// TIA Portal project "Projec1214" (V17)

(* hardware
DEVICE "S7-1200 station_1"  S7-1200 Station
   slot 0: "Rack_0"  S7-1200 Rack  Rack  V1.0
   slot 1: "PLC_1"  CPU 1211C DC/DC/Rly  6ES7 211-1HE40-0XB0  V4.5
DEVICE "HMI_1"  KTP400 Comfort
   slot 0: "HMI_1"  KTP400 Comfort  6AV2 124-2DC01-0AX0  17.0.0.0
   slot 1: "HMI_RT_1"  KTP400 Comfort  6AV2 124-2DC01-0AX0  17.0.0.0
   slot 5: "HMI_1.IE_CP_1"  PROFINET Interface  17.0.0.0
      slot 1: "PROFINET Interface_1"  PROFINET Interface
         slot 1: "Port_1"  Port
   slot 7: "HMI_1.MPI/DP_CP_1"  MPI/DP Interface  17.0.0.0
*)

// ===== PLC "PLC_1"  CPU 1211C DC/DC/Rly =====

VAR_GLOBAL   // PLC tag table "Default tag table"
   "BP_Appel_ET1" AT %I0.1 : Bool;
   "BP_Appel_ET2" AT %I0.2 : Bool;
   "BP_Appel_ET3" AT %I0.3 : Bool;
   "Position_ET1" AT %I0.5 : Bool;
   "Position_ET2" AT %I0.6 : Bool;
   "Position_ET3" AT %I0.7 : Bool;
   "Monter" AT %Q0.0 : Bool;
   "Descente" AT %Q0.1 : Bool;
   "Ouverture" AT %Q0.2 : Bool;
   "Fermeture" AT %Q0.3 : Bool;
   "MemoAppelET1" AT %M10.1 : Bool;
   "MemoAppelET2" AT %M10.2 : Bool;
   "MemoAppelET3" AT %M10.3 : Bool;
   "ETAPE0" AT %M10.4 : Bool;
   "ETAPE1" AT %M10.5 : Bool;
   "ETAPE2" AT %M10.6 : Bool;
   "ETAPE3" AT %M10.7 : Bool;
   "ETAPE4" AT %M11.0 : Bool;
   "ETAPE5" AT %M11.1 : Bool;
   "ETAPE6" AT %M11.2 : Bool;
   "ETAPE7" AT %M11.3 : Bool;
   "ETAPE8" AT %M11.4 : Bool;
   "ETAPE9" AT %M11.5 : Bool;
   "PorteOuverte" AT %I1.0 : Bool;
   "PorteFermee" AT %I1.1 : Bool;
   "MemoPosiET1" AT %M11.6 : Bool;
   "MemoPosiET2" AT %M11.7 : Bool;
   "MemoPosiET3" AT %M12.0 : Bool;
   "MemoPorteOuverte" AT %M12.1 : Bool;
   "MemoPorteFermee" AT %M12.2 : Bool;
   "DemandeNiveau1" AT %M40.0 : Bool;
   "DemandeNIveau2" AT %M40.1 : Bool;
   "DemandeNiveau3" AT %M40.2 : Bool;
   "Tag_4" AT %M40.3 : Bool;
   "Tag_5" AT %M40.4 : Bool;
   "Tag_6" AT %M40.5 : Bool;
   "Tag_7" AT %M40.6 : Bool;
   "Tag_8" AT %M40.7 : Bool;
   "deplacemntAsceseur" AT %MW100 : Int;
   "DeplacementPorteG" AT %MW102 : Int;
   "DeplacementPorteD" AT %MW104 : Int;
   "Clock_Byte" AT %MB0 : Byte;
   "Clock_10Hz" AT %M0.0 : Bool;
   "Clock_5Hz" AT %M0.1 : Bool;
   "Clock_2.5Hz" AT %M0.2 : Bool;
   "Clock_2Hz" AT %M0.3 : Bool;
   "Clock_1.25Hz" AT %M0.4 : Bool;
   "Clock_1Hz" AT %M0.5 : Bool;
   "Clock_0.625Hz" AT %M0.6 : Bool;
   "Clock_0.5Hz" AT %M0.7 : Bool;
   "deplacementHautPorte" AT %MW106 : Int;
END_VAR

DATA_BLOCK "ETAPE"   // DB1
{ S7_Optimized_Access := 'TRUE' }
VERSION : 0.1
   VAR
      "1" : Bool;
      "0" : Bool;
      "2" : Bool;
      "3" : Bool;
      "6" : Bool;
      "7" : Bool;
      "8" : Bool;
   END_VAR
BEGIN
END_DATA_BLOCK

// folder: System blocks/Program resources

DATA_BLOCK "IEC_Timer_0_DB"   // DB2
{ S7_Optimized_Access := 'TRUE' }
AUTHOR : Simatic
FAMILY : IEC
NAME : IEC_TMR
VERSION : 1.0
// stored: InstanceOfName IEC_TIMER
"IEC_TIMER"
BEGIN
END_DATA_BLOCK

// folder: (top level)

ORGANIZATION_BLOCK "Main"   // OB1, LAD, ProgramCycle
TITLE = "Main Program Sweep (Cycle)"
{ S7_Optimized_Access := 'TRUE' }
VERSION : 0.1
   VAR_INPUT
      Initial_Call : Bool;   // Initial call of this OB
      Remanence : Bool;   // =True, if remanent data are available
   END_VAR
   VAR_TEMP   // added for the SCL form of the ladder/FBD networks
      _w1 : Bool;
   END_VAR
BEGIN

REGION Network 1: ETAPE0
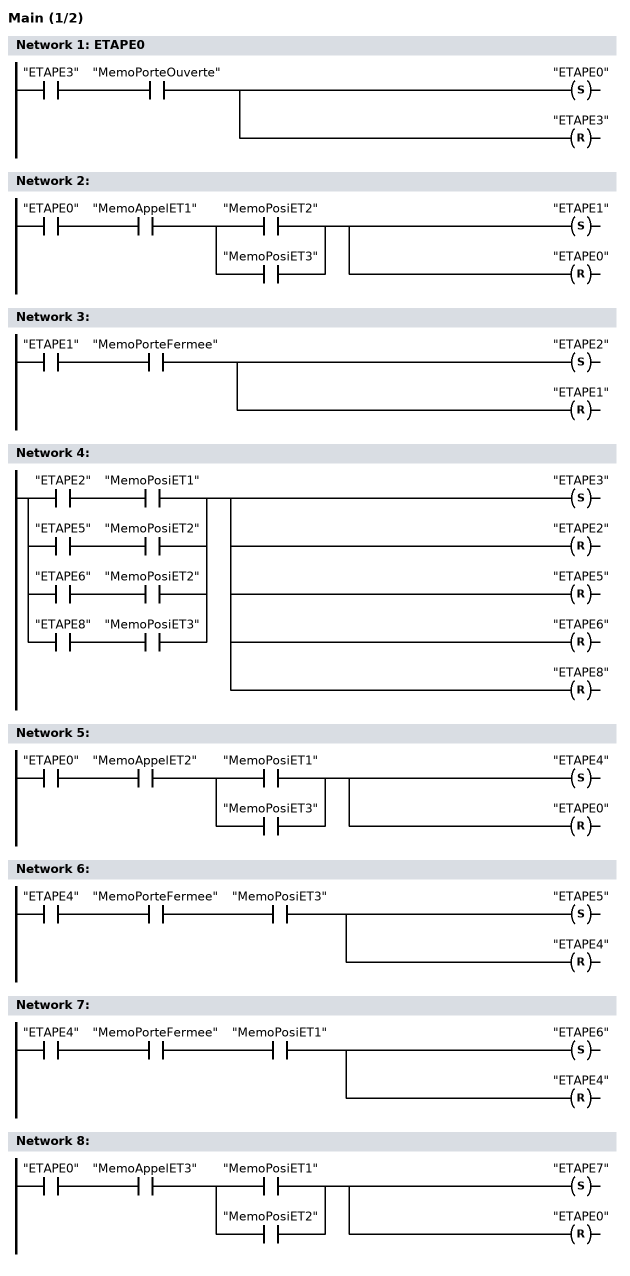
   RUNG wire#powerrail
      Contact( "ETAPE3" )
      Contact( "MemoPorteOuverte" )
      wire#w1
      S_Coil( "ETAPE0" )
   END_RUNG
   RUNG wire#w1
      R_Coil( "ETAPE3" )
   END_RUNG
   // the same network as SCL:
   IF "ETAPE3" AND "MemoPorteOuverte" THEN
       "ETAPE0" := TRUE;
       "ETAPE3" := FALSE;
   END_IF;
END_REGION

REGION Network 2
   RUNG wire#powerrail
      Contact( "ETAPE0" )
      Contact( "MemoAppelET1" )
      wire#w1
      Contact( "MemoPosiET2" )
      wire#w2
      S_Coil( "ETAPE1" )
   END_RUNG
   RUNG wire#w1
      Contact( "MemoPosiET3" )
   END_RUNG wire#w2
   RUNG wire#w2
      R_Coil( "ETAPE0" )
   END_RUNG
   // the same network as SCL:
   IF "ETAPE0" AND "MemoAppelET1" AND ("MemoPosiET2" OR "MemoPosiET3") THEN
       "ETAPE1" := TRUE;
       "ETAPE0" := FALSE;
   END_IF;
END_REGION

REGION Network 3
   RUNG wire#powerrail
      Contact( "ETAPE1" )
      Contact( "MemoPorteFermee" )
      wire#w1
      S_Coil( "ETAPE2" )
   END_RUNG
   RUNG wire#w1
      R_Coil( "ETAPE1" )
   END_RUNG
   // the same network as SCL:
   IF "ETAPE1" AND "MemoPorteFermee" THEN
       "ETAPE2" := TRUE;
       "ETAPE1" := FALSE;
   END_IF;
END_REGION

REGION Network 4
   RUNG wire#powerrail
      Contact( "ETAPE2" )
      Contact( "MemoPosiET1" )
      wire#w1
      S_Coil( "ETAPE3" )
   END_RUNG
   RUNG wire#powerrail
      Contact( "ETAPE5" )
      Contact( "MemoPosiET2" )
   END_RUNG wire#w1
   RUNG wire#powerrail
      Contact( "ETAPE6" )
      Contact( "MemoPosiET2" )
   END_RUNG wire#w1
   RUNG wire#powerrail
      Contact( "ETAPE8" )
      Contact( "MemoPosiET3" )
   END_RUNG wire#w1
   RUNG wire#w1
      R_Coil( "ETAPE2" )
   END_RUNG
   RUNG wire#w1
      R_Coil( "ETAPE5" )
   END_RUNG
   RUNG wire#w1
      R_Coil( "ETAPE6" )
   END_RUNG
   RUNG wire#w1
      R_Coil( "ETAPE8" )
   END_RUNG
   // the same network as SCL:
   IF ("ETAPE2" AND "MemoPosiET1") OR ("ETAPE5" AND "MemoPosiET2") OR ("ETAPE6" AND "MemoPosiET2") OR ("ETAPE8" AND "MemoPosiET3") THEN
       "ETAPE3" := TRUE;
   END_IF;
   #_w1 := ("ETAPE2" AND "MemoPosiET1") OR ("ETAPE5" AND "MemoPosiET2") OR ("ETAPE6" AND "MemoPosiET2") OR ("ETAPE8" AND "MemoPosiET3");
   IF #_w1 THEN
       "ETAPE2" := FALSE;
       "ETAPE5" := FALSE;
       "ETAPE6" := FALSE;
       "ETAPE8" := FALSE;
   END_IF;
END_REGION

REGION Network 5
   RUNG wire#powerrail
      Contact( "ETAPE0" )
      Contact( "MemoAppelET2" )
      wire#w1
      Contact( "MemoPosiET1" )
      wire#w2
      S_Coil( "ETAPE4" )
   END_RUNG
   RUNG wire#w1
      Contact( "MemoPosiET3" )
   END_RUNG wire#w2
   RUNG wire#w2
      R_Coil( "ETAPE0" )
   END_RUNG
   // the same network as SCL:
   IF "ETAPE0" AND "MemoAppelET2" AND ("MemoPosiET1" OR "MemoPosiET3") THEN
       "ETAPE4" := TRUE;
       "ETAPE0" := FALSE;
   END_IF;
END_REGION

REGION Network 6
   RUNG wire#powerrail
      Contact( "ETAPE4" )
      Contact( "MemoPorteFermee" )
      Contact( "MemoPosiET3" )
      wire#w1
      S_Coil( "ETAPE5" )
   END_RUNG
   RUNG wire#w1
      R_Coil( "ETAPE4" )
   END_RUNG
   // the same network as SCL:
   IF "ETAPE4" AND "MemoPorteFermee" AND "MemoPosiET3" THEN
       "ETAPE5" := TRUE;
       "ETAPE4" := FALSE;
   END_IF;
END_REGION

REGION Network 7
   RUNG wire#powerrail
      Contact( "ETAPE4" )
      Contact( "MemoPorteFermee" )
      Contact( "MemoPosiET1" )
      wire#w1
      S_Coil( "ETAPE6" )
   END_RUNG
   RUNG wire#w1
      R_Coil( "ETAPE4" )
   END_RUNG
   // the same network as SCL:
   IF "ETAPE4" AND "MemoPorteFermee" AND "MemoPosiET1" THEN
       "ETAPE6" := TRUE;
       "ETAPE4" := FALSE;
   END_IF;
END_REGION

REGION Network 8
   RUNG wire#powerrail
      Contact( "ETAPE0" )
      Contact( "MemoAppelET3" )
      wire#w1
      Contact( "MemoPosiET1" )
      wire#w2
      S_Coil( "ETAPE7" )
   END_RUNG
   RUNG wire#w1
      Contact( "MemoPosiET2" )
   END_RUNG wire#w2
   RUNG wire#w2
      R_Coil( "ETAPE0" )
   END_RUNG
   // the same network as SCL:
   IF "ETAPE0" AND "MemoAppelET3" AND ("MemoPosiET1" OR "MemoPosiET2") THEN
       "ETAPE7" := TRUE;
       "ETAPE0" := FALSE;
   END_IF;
END_REGION

REGION Network 9
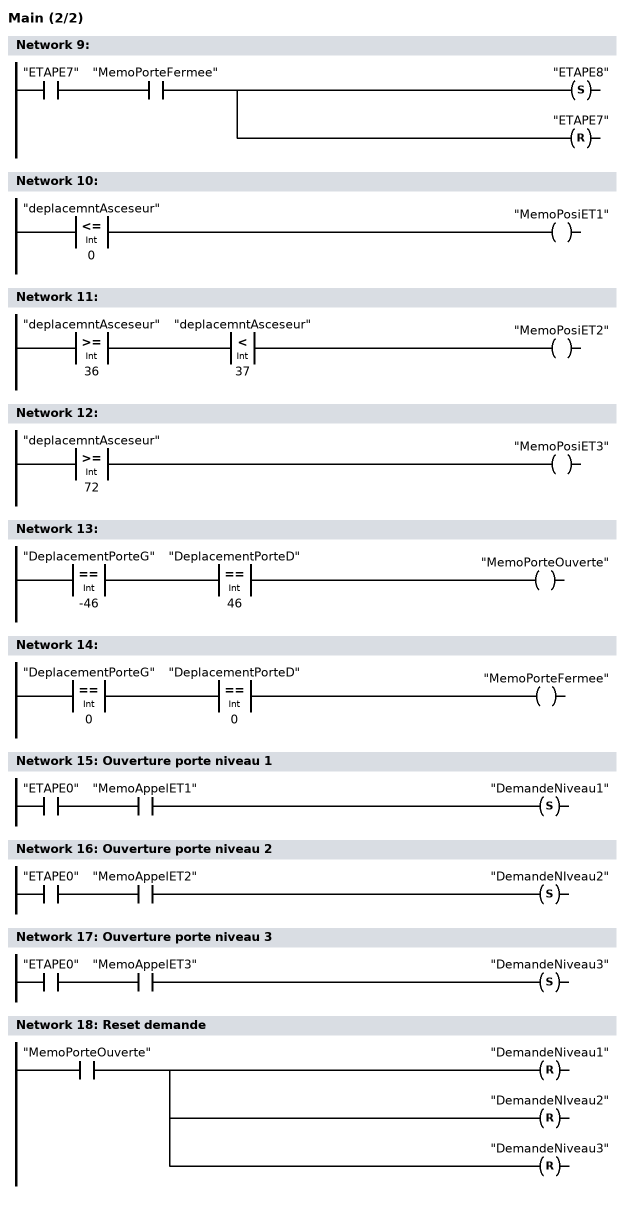
   RUNG wire#powerrail
      Contact( "ETAPE7" )
      Contact( "MemoPorteFermee" )
      wire#w1
      S_Coil( "ETAPE8" )
   END_RUNG
   RUNG wire#w1
      R_Coil( "ETAPE7" )
   END_RUNG
   // the same network as SCL:
   IF "ETAPE7" AND "MemoPorteFermee" THEN
       "ETAPE8" := TRUE;
       "ETAPE7" := FALSE;
   END_IF;
END_REGION

REGION Network 10
   RUNG wire#powerrail
      { S7_Templates := "SrcType := Int" } LE_Contact(in1 := "deplacemntAsceseur", in2 := 0)
      Coil( "MemoPosiET1" )
   END_RUNG
   // the same network as SCL:
   "MemoPosiET1" := "deplacemntAsceseur" <= 0;
END_REGION

REGION Network 11
   RUNG wire#powerrail
      { S7_Templates := "SrcType := Int" } GE_Contact(in1 := "deplacemntAsceseur", in2 := 36)
      { S7_Templates := "SrcType := Int" } LT_Contact(in1 := "deplacemntAsceseur", in2 := 37)
      Coil( "MemoPosiET2" )
   END_RUNG
   // the same network as SCL:
   "MemoPosiET2" := ("deplacemntAsceseur" >= 36) AND ("deplacemntAsceseur" < 37);
END_REGION

REGION Network 12
   RUNG wire#powerrail
      { S7_Templates := "SrcType := Int" } GE_Contact(in1 := "deplacemntAsceseur", in2 := 72)
      Coil( "MemoPosiET3" )
   END_RUNG
   // the same network as SCL:
   "MemoPosiET3" := "deplacemntAsceseur" >= 72;
END_REGION

REGION Network 13
   RUNG wire#powerrail
      { S7_Templates := "SrcType := Int" } EQ_Contact(in1 := "DeplacementPorteG", in2 := -46)
      { S7_Templates := "SrcType := Int" } EQ_Contact(in1 := "DeplacementPorteD", in2 := 46)
      Coil( "MemoPorteOuverte" )
   END_RUNG
   // the same network as SCL:
   "MemoPorteOuverte" := ("DeplacementPorteG" = (-46)) AND ("DeplacementPorteD" = 46);
END_REGION

REGION Network 14
   RUNG wire#powerrail
      { S7_Templates := "SrcType := Int" } EQ_Contact(in1 := "DeplacementPorteG", in2 := 0)
      { S7_Templates := "SrcType := Int" } EQ_Contact(in1 := "DeplacementPorteD", in2 := 0)
      Coil( "MemoPorteFermee" )
   END_RUNG
   // the same network as SCL:
   "MemoPorteFermee" := ("DeplacementPorteG" = 0) AND ("DeplacementPorteD" = 0);
END_REGION

REGION Network 15: Ouverture porte niveau 1
   RUNG wire#powerrail
      Contact( "ETAPE0" )
      Contact( "MemoAppelET1" )
      S_Coil( "DemandeNiveau1" )
   END_RUNG
   // the same network as SCL:
   IF "ETAPE0" AND "MemoAppelET1" THEN "DemandeNiveau1" := TRUE; END_IF;
END_REGION

REGION Network 16: Ouverture porte niveau 2
   RUNG wire#powerrail
      Contact( "ETAPE0" )
      Contact( "MemoAppelET2" )
      S_Coil( "DemandeNIveau2" )
   END_RUNG
   // the same network as SCL:
   IF "ETAPE0" AND "MemoAppelET2" THEN "DemandeNIveau2" := TRUE; END_IF;
END_REGION

REGION Network 17: Ouverture porte niveau 3
   RUNG wire#powerrail
      Contact( "ETAPE0" )
      Contact( "MemoAppelET3" )
      S_Coil( "DemandeNiveau3" )
   END_RUNG
   // the same network as SCL:
   IF "ETAPE0" AND "MemoAppelET3" THEN "DemandeNiveau3" := TRUE; END_IF;
END_REGION

REGION Network 18: Reset demande
   RUNG wire#powerrail
      Contact( "MemoPorteOuverte" )
      wire#w1
      R_Coil( "DemandeNiveau1" )
   END_RUNG
   RUNG wire#w1
      R_Coil( "DemandeNIveau2" )
   END_RUNG
   RUNG wire#w1
      R_Coil( "DemandeNiveau3" )
   END_RUNG
   // the same network as SCL:
   IF "MemoPorteOuverte" THEN
       "DemandeNiveau1" := FALSE;
       "DemandeNIveau2" := FALSE;
       "DemandeNiveau3" := FALSE;
   END_IF;
END_REGION
END_ORGANIZATION_BLOCK

ORGANIZATION_BLOCK "Cyclic interrupt"   // OB30, LAD, CyclicInterrupt
{ S7_Optimized_Access := 'TRUE' }
VERSION : 0.1
   VAR_INPUT
      Initial_Call : Bool;   // Initial call of this OB
      Event_Count : Int;   // Events discarded
   END_VAR
   VAR_TEMP   // added for the SCL form of the ladder/FBD networks
      _w1 : Bool;
   END_VAR
BEGIN

REGION Network 1: Fermeture porte
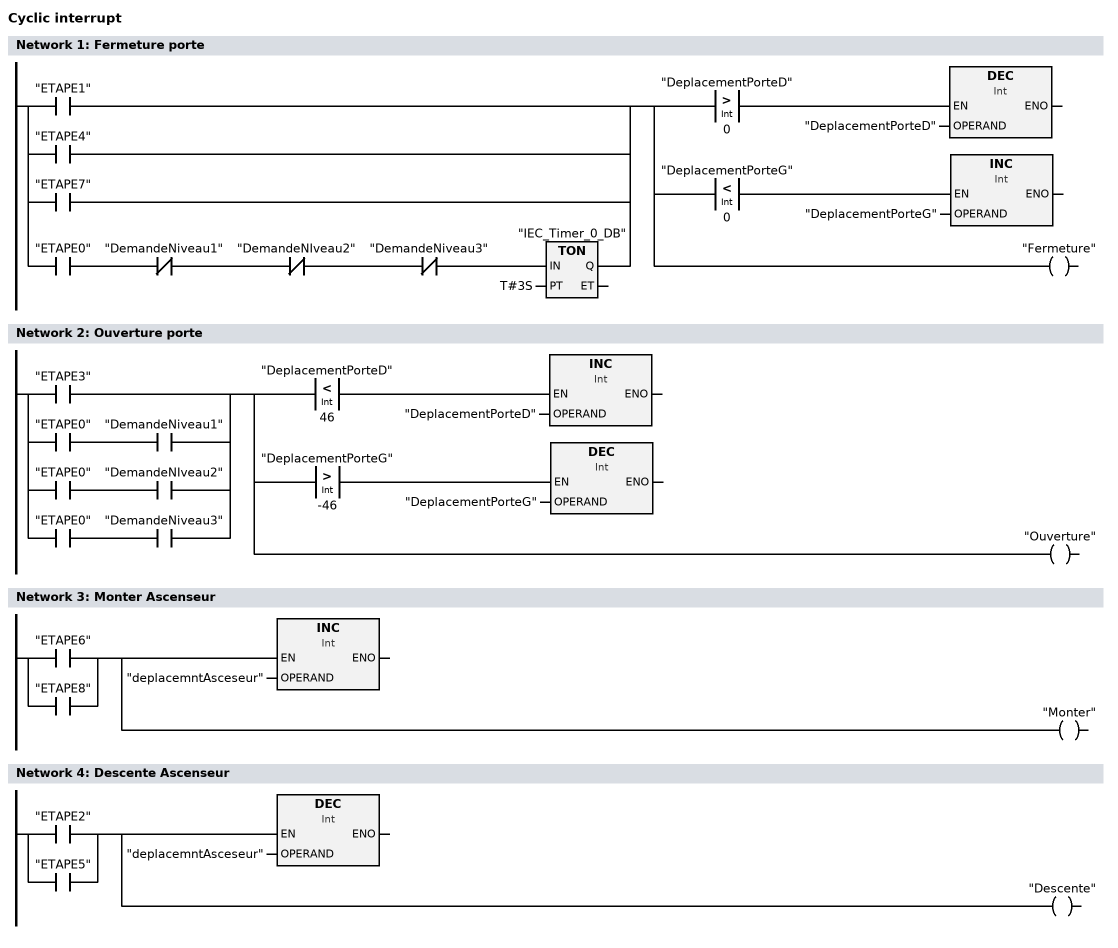
   "IEC_Timer_0_DB".TON(IN := "ETAPE0" AND NOT "DemandeNiveau1" AND NOT "DemandeNIveau2" AND NOT "DemandeNiveau3",
                        PT := T#3S);
   #_w1 := "ETAPE1" OR "ETAPE4" OR "ETAPE7" OR "IEC_Timer_0_DB".Q;
   IF #_w1 AND ("DeplacementPorteD" > 0) THEN "DeplacementPorteD" := "DeplacementPorteD" - 1; END_IF;
   IF #_w1 AND ("DeplacementPorteG" < 0) THEN "DeplacementPorteG" := "DeplacementPorteG" + 1; END_IF;
   "Fermeture" := #_w1;
END_REGION

REGION Network 2: Ouverture porte
   RUNG wire#powerrail
      Contact( "ETAPE3" )
      wire#w1
      { S7_Templates := "SrcType := Int" } LT_Contact(in1 := "DeplacementPorteD", in2 := 46)
      { S7_Templates := "DestType := Int" } Inc( "DeplacementPorteD" )
   END_RUNG
   RUNG wire#powerrail
      Contact( "ETAPE0" )
      Contact( "DemandeNiveau1" )
   END_RUNG wire#w1
   RUNG wire#powerrail
      Contact( "ETAPE0" )
      Contact( "DemandeNIveau2" )
   END_RUNG wire#w1
   RUNG wire#powerrail
      Contact( "ETAPE0" )
      Contact( "DemandeNiveau3" )
   END_RUNG wire#w1
   RUNG wire#w1
      { S7_Templates := "SrcType := Int" } GT_Contact(in1 := "DeplacementPorteG", in2 := -46)
      { S7_Templates := "DestType := Int" } Dec( "DeplacementPorteG" )
   END_RUNG
   RUNG wire#w1
      Coil( "Ouverture" )
   END_RUNG
   // the same network as SCL:
   #_w1 := "ETAPE3" OR ("ETAPE0" AND "DemandeNiveau1") OR ("ETAPE0" AND "DemandeNIveau2") OR ("ETAPE0" AND "DemandeNiveau3");
   IF #_w1 AND ("DeplacementPorteD" < 46) THEN "DeplacementPorteD" := "DeplacementPorteD" + 1; END_IF;
   IF #_w1 AND ("DeplacementPorteG" > (-46)) THEN "DeplacementPorteG" := "DeplacementPorteG" - 1; END_IF;
   "Ouverture" := #_w1;
END_REGION

REGION Network 3: Monter Ascenseur
   RUNG wire#powerrail
      Contact( "ETAPE6" )
      wire#w1
      { S7_Templates := "DestType := Int" } Inc( "deplacemntAsceseur" )
   END_RUNG
   RUNG wire#powerrail
      Contact( "ETAPE8" )
   END_RUNG wire#w1
   RUNG wire#w1
      Coil( "Monter" )
   END_RUNG
   // the same network as SCL:
   #_w1 := "ETAPE6" OR "ETAPE8";
   IF #_w1 THEN "deplacemntAsceseur" := "deplacemntAsceseur" + 1; END_IF;
   "Monter" := #_w1;
END_REGION

REGION Network 4: Descente Ascenseur
   RUNG wire#powerrail
      Contact( "ETAPE2" )
      wire#w1
      { S7_Templates := "DestType := Int" } Dec( "deplacemntAsceseur" )
   END_RUNG
   RUNG wire#powerrail
      Contact( "ETAPE5" )
   END_RUNG wire#w1
   RUNG wire#w1
      Coil( "Descente" )
   END_RUNG
   // the same network as SCL:
   #_w1 := "ETAPE2" OR "ETAPE5";
   IF #_w1 THEN "deplacemntAsceseur" := "deplacemntAsceseur" - 1; END_IF;
   "Descente" := #_w1;
END_REGION
END_ORGANIZATION_BLOCK

ORGANIZATION_BLOCK "Startup"   // OB100, LAD, Startup
TITLE = "Complete Restart"
{ S7_Optimized_Access := 'TRUE' }
VERSION : 0.1
   VAR_INPUT
      LostRetentive : Bool;   // True if retentive data are lost
      LostRTC : Bool;   // True if date and time are lost
   END_VAR
BEGIN

REGION Network 1
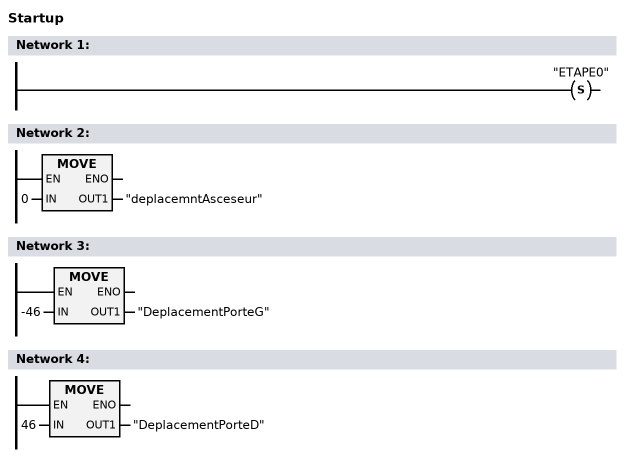
   RUNG wire#powerrail
      S_Coil( "ETAPE0" )
   END_RUNG
   // the same network as SCL:
   "ETAPE0" := TRUE;
END_REGION

REGION Network 2
   RUNG wire#powerrail
      Move(in := 0, out1 => "deplacemntAsceseur")
   END_RUNG
   // the same network as SCL:
   "deplacemntAsceseur" := 0;
END_REGION

REGION Network 3
   RUNG wire#powerrail
      Move(in := -46, out1 => "DeplacementPorteG")
   END_RUNG
   // the same network as SCL:
   "DeplacementPorteG" := -46;
END_REGION

REGION Network 4
   RUNG wire#powerrail
      Move(in := 46, out1 => "DeplacementPorteD")
   END_RUNG
   // the same network as SCL:
   "DeplacementPorteD" := 46;
END_REGION
END_ORGANIZATION_BLOCK

(* ===== HMI "HMI_RT_1" =====
system functions are stored by id; their names below are inferred from use
connection "HMI_Connection_1": ETHERNET, S7_1200_OMS

HMI tags "Default tag table"
   "ETAPE0" : Bool = PLC ETAPE0 AT %M10.4, 1 s
   "ETAPE1" : Bool = PLC ETAPE1 AT %M10.5, 1 s
   "ETAPE2" : Bool = PLC ETAPE2 AT %M10.6, 1 s
   "ETAPE3" : Bool = PLC ETAPE3 AT %M10.7, 1 s
   "ETAPE4" : Bool = PLC ETAPE4 AT %M11.0, 1 s
   "ETAPE5" : Bool = PLC ETAPE5 AT %M11.1, 1 s
   "ETAPE6" : Bool = PLC ETAPE6 AT %M11.2, 1 s
   "ETAPE7" : Bool = PLC ETAPE7 AT %M11.3, 1 s
   "ETAPE8" : Bool = PLC ETAPE8 AT %M11.4, 1 s
   "deplacemntAsceseur" : Int = PLC deplacemntAsceseur AT %MW100, 1 s
   "DeplacementPorteG" : Int = PLC DeplacementPorteG AT %MW102, 1 s
   "DeplacementPorteD" : Int = PLC DeplacementPorteD AT %MW104, 1 s
   "MemoAppelET1" : Bool = PLC MemoAppelET1 AT %M10.1, 1 s
   "MemoAppelET2" : Bool = PLC MemoAppelET2 AT %M10.2, 1 s
   "MemoAppelET3" : Bool = PLC MemoAppelET3 AT %M10.3, 1 s
   "Position_ET1" : Bool = PLC Position_ET1 AT %I0.5, 1 s
   "Position_ET2" : Bool = PLC Position_ET2 AT %I0.6, 1 s
   "Position_ET3" : Bool = PLC Position_ET3 AT %I0.7, 1 s
   "MemoPosiET1" : Bool = PLC MemoPosiET1 AT %M11.6, 1 s
   "MemoPosiET2" : Bool = PLC MemoPosiET2 AT %M11.7, 1 s
   "MemoPosiET3" : Bool = PLC MemoPosiET3 AT %M12.0, 1 s
   "deplacementHautPorte" : Int = PLC deplacementHautPorte AT %MW106, 1 s

screen "Vue grafcet" 480x272, template "Template_1"
   Button "Button_1" at 363,241 size 117x31; TextOff 'Vue Ascenseur'
      on Press: ActivateScreen("Vue ascenseur", 0)
   Rectangle "Rectangle_1" at 186,230 size 49x42
      Appearance <- "ETAPE3"
   Rectangle "Rectangle_2" at 187,10 size 49x42
      Appearance <- "ETAPE0"
   Rectangle "Rectangle_3" at 397,80 size 49x42
      Appearance <- "ETAPE7"
   Rectangle "Rectangle_4" at 186,80 size 49x42
      Appearance <- "ETAPE4"
   Rectangle "Rectangle_5" at 17,80 size 49x42
      Appearance <- "ETAPE1"
   Rectangle "Rectangle_6" at 397,158 size 49x42
      Appearance <- "ETAPE8"
   Rectangle "Rectangle_7" at 276,160 size 49x42
      Appearance <- "ETAPE6"
   Rectangle "Rectangle_8" at 100,160 size 49x42
      Appearance <- "ETAPE5"
   Rectangle "Rectangle_9" at 18,158 size 49x42
      Appearance <- "ETAPE2"
   TextField "Text field_1" at 199,20 size 30x20; Text 'ET0'
   TextField "Text field_3" at 199,240 size 30x20; Text 'ET3'
   TextField "Text field_4" at 26,168 size 30x20; Text 'ET2'
   TextField "Text field_5" at 109,168 size 30x20; Text 'ET5'
   TextField "Text field_6" at 408,168 size 30x20; Text 'ET8'
   TextField "Text field_7" at 289,168 size 30x20; Text 'ET6'
   TextField "Text field_8" at 30,91 size 30x20; Text 'ET1'
   TextField "Text field_9" at 200,91 size 30x20; Text 'ET4'
   TextField "Text field_10" at 409,88 size 30x20; Text 'ET7'

screen "Vue ascenseur" 480x272
   Button "Button_1" at 384,240 size 96x32; TextOff 'Vue grafcet'
      on Press: ActivateScreen("Vue grafcet", 0)
   TextField "Text field_1" at 16,238 size 14x20; Text '1'
   TextField "Text field_2" at 18,160 size 14x20; Text '2'
   TextField "Text field_3" at 13,90 size 14x20; Text '3'
   Button "Button_4" at 210,232 size 76x32; TextOff 'P1'
      on Press: function_b14e0dd5("MemoAppelET1", 0)
      Appearance <- "MemoPosiET1"
   Button "Button_2" at 210,156 size 78x33; TextOff 'P2'
      on Press: function_b14e0dd5("MemoAppelET2", 0)
      Appearance <- "MemoPosiET2"
   Button "Button_3" at 219,71 size 75x29; TextOff 'P3'
      on Press: function_b14e0dd5("MemoAppelET3", 0)
      Appearance <- "MemoPosiET3"
   IOField "I/O field_1" at 239,3 size 96x32; FormatPattern s99999
      ProcessValue <- "deplacementHautPorte"
   Group "Group" at 48,200 size 100x71
      VerticalMovement <- "deplacemntAsceseur"
   Rectangle "Rectangle_2" at 100,200 size 46x70
      DirectMovement <- "DeplacementPorteD"
      DirectMovement <- "deplacementHautPorte"
   Rectangle "Rectangle_3" at 50,200 size 46x70
      DirectMovement <- "DeplacementPorteG"
*)